// TIA Portal V18 export
// export: Created 2026-06-08T17:01:58.4945456Z, ExportSetting WithDefaults, DisplayName Totally Integrated Automation Portal, DisplayVersion V18, DisplayName TIA Portal Openness, DisplayVersion V18, DisplayName TIA Portal Version Control Interface, DisplayVersion V18, DisplayName STEP 7 Professional, DisplayVersion V18, DisplayName STEP 7 Safety, DisplayVersion V18, DisplayName WinCC Professional, DisplayVersion V18
DATA_BLOCK "M1_MOTOR_DB"   // DB8
VERSION : 0.1
// stored: AutoNumber true, DBAccessibleFromOPCUA true, InstanceOfName M1_MOTOR, InstanceOfType FB
"M1_MOTOR"
   // VAR_INPUT
   //    EMERGENCY_STATE : Bool;
   //    WIND_DOWN : Bool;
   //    INTERLOCK_R : Bool;
   //    MOVE_R : Bool;
   //    INTERLOCK_F : Bool;
   //    MOVE_F : Bool;
   //    COIL_F : Bool;
   //    TRIP_COUNT_FINISHED : Bool;
   // END_VAR
   // VAR_OUTPUT
   //    COIL_R_OUT : Bool;
   //    COIL_R_OUT_HMI : Bool;
   //    COIL_F_OUT : Bool;
   //    COIL_F_OUT_HMI : Bool;
   // END_VAR
BEGIN
END_DATA_BLOCK
